// TIA Portal V18 export
FUNCTION "RTG2_POST" : Void   // FC15, LAD
{ S7_Optimized_Access := 'TRUE' }
// stored: SetENOAutomatically false
BEGIN

REGION Network 1: Send the data to RTG1
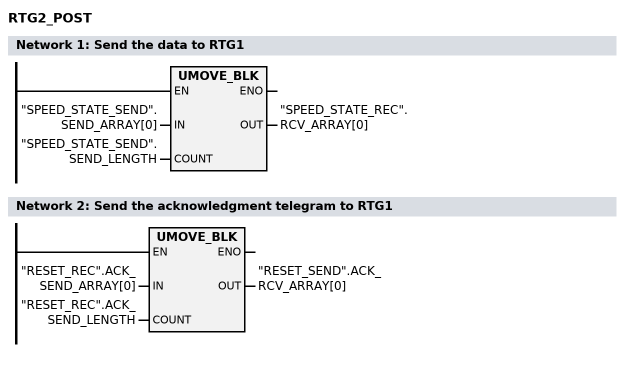
   UMOVE_BLK(IN := "SPEED_STATE_SEND".SEND_ARRAY[0],
             COUNT := "SPEED_STATE_SEND".SEND_LENGTH,
             OUT => "SPEED_STATE_REC".RCV_ARRAY[0]);
END_REGION

REGION Network 2: Send the acknowledgment telegram to RTG1
   UMOVE_BLK(IN := "RESET_REC".ACK_SEND_ARRAY[0],
             COUNT := "RESET_REC".ACK_SEND_LENGTH,
             OUT => "RESET_SEND".ACK_RCV_ARRAY[0]);
END_REGION
END_FUNCTION
